{attribute 'GeneratedUsingTerminal: EK1100-0000-0018'}
{attribute addProperty BoxType "EK1100-0000-0018"}
{attribute addProperty Id "Beckhoff_EPP2xxxEK1122Beckhoff_EPP2xxxEK1122_A0F3DD5A1956"}
{attribute addProperty CRC "3433037725"}
{attribute addProperty Size "1956"}
TYPE Beckhoff_EPP2xxx_CC9FFF9D EXTENDS EK1100_1FC0878B :
STRUCT
	{attribute addProperty Name "Beckhoff_EPP2xxxEK1122"}
	{attribute addProperty PreviousPort "Beckhoff EPP2xxx : B"}
	Beckhoff_EPP2xxxEK1122 : Beckhoff_EPP2xxxEK1122_A0F3DD5A;
END_STRUCT
END_TYPE

(* stored: Version 1.2.0.0, ProductVersion 3.1.4024.9
   DUT Beckhoff_EPP2xxx_CC9FFF9D: Id {0630ce9d-25c5-4117-92c4-043261ace1eb} *)
